Universal Robots PolyScope program: punto3_pickplace_NEW.urp

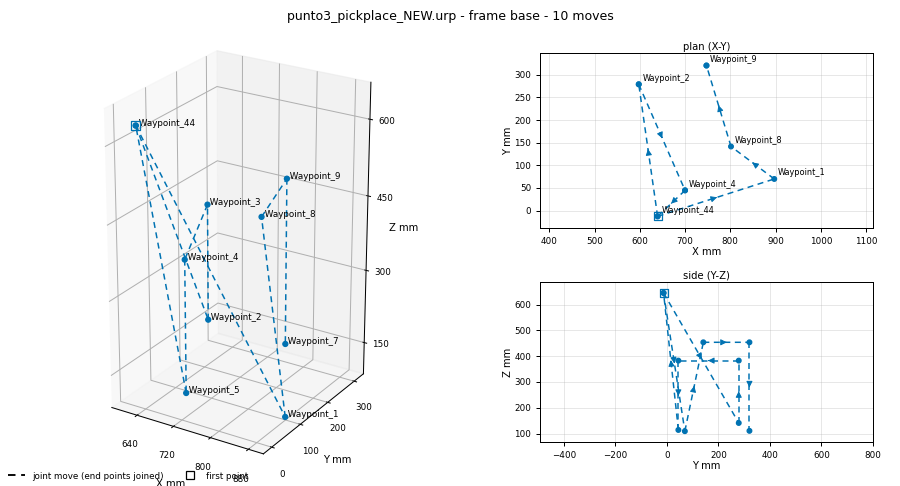
[picture p0: tool path of punto3_pickplace_NEW.urp in frame base, 10 of 10 moves have a stored position in this frame; points joined in program order, loops and branches not executed]
Program punto3_pickplace (installation=default directory=/ursim/programs createdIn=3.15.8.106339 lastSavedIn=3.15.8.106339 robotSerialNumber=2018359999)
Calibrated DH parameters: a=[0, -0.425, -0.39225, 0, 0, 0]; d=[0.089159, 0, 0, 0.10915, 0.09465, 0.0823]; alpha=[1.570796, 0, 0, 1.570796, -1.570796, 0]; deltaTheta=[0, 0, 0, 0, 0, 0]
Robot Program (runOnlyOnce=false)
  MoveJ speed 60 deg/s, acceleration 80 deg/s^2 (useActiveTCP=true)
    Set DigitalOutput pin=digital_out[0]; digitalValue=0
    Waypoint Waypoint_44: TCP in base x=639.374 y=-12.799 z=645.611 mm, rx=2.7019 ry=1.4477 rz=0.2985 rad; joints [8.631, -138.345, 17.122, 222.891, 90.378, -137.696] deg
    Wait DigitalInput pin=digital_in[0]; digitalValue=1
    Wait Sleep waitTime=2
    Waypoint Waypoint_2: TCP in base x=597.72 y=279.007 z=140.951 mm, rx=2.7019 ry=1.4477 rz=0.2985 rad; joints [35.16, -123.066, -94.887, 318.588, 85.157, -111.657] deg
    Set DigitalOutput pin=digital_out[0]; digitalValue=1
    Popup Message (haltProgram=false message=se cerró el gripper  inputType=Text)
    Waypoint Waypoint_3: TCP in base x=597.72 y=279.007 z=383.015 mm, rx=2.7019 ry=1.4477 rz=0.2985 rad; joints [35.16, -110.812, -75.083, 286.529, 85.157, -111.657] deg
    Popup Message (haltProgram=false message=punto intermedio principal inputType=Text)
    Wait Sleep waitTime=1
    Waypoint Waypoint_4: TCP in base x=700.042 y=44.656 z=383.015 mm, rx=2.7019 ry=1.4477 rz=0.2985 rad; joints [12.653, -116.851, -66.636, 285.153, 89.564, -133.757] deg
    Popup Message (haltProgram=false message=punto intermedio secundario inputType=Text)
    Wait Sleep waitTime=1
    Waypoint Waypoint_5: TCP in base x=700.042 y=44.656 z=113.852 mm, rx=2.7019 ry=1.4477 rz=0.2985 rad; joints [12.653, -129.957, -87.698, 319.32, 89.564, -133.757] deg
    Set DigitalOutput pin=digital_out[0]; digitalValue=0
    Popup Message (haltProgram=false message=se abrió el gripper inputType=Text)
    Waypoint Waypoint_44: TCP in base x=639.374 y=-12.799 z=645.611 mm, rx=2.7019 ry=1.4477 rz=0.2985 rad; joints [8.631, -138.345, 17.122, 222.891, 90.378, -137.696] deg
    Wait Sleep waitTime=2
    Waypoint Waypoint_1: TCP in base x=897.17 y=69.826 z=109 mm, rx=2.7019 ry=1.4477 rz=0.2985 rad; joints [11.435, -159.34, -30.741, 291.753, 89.811, -134.95] deg
    Set DigitalOutput pin=digital_out[0]; digitalValue=1
    Popup Message (haltProgram=false message=se cerró el gripper inputType=Text)
    Waypoint Waypoint_8: TCP in base x=801.574 y=141.533 z=454.057 mm, rx=2.7019 ry=1.4477 rz=0.2985 rad; joints [17.872, -148.017, -1.091, 250.688, 88.512, -128.645] deg
    Popup Message (haltProgram=false message=punto intermedio inicial inputType=Text)
    Waypoint Waypoint_9: TCP in base x=747.352 y=320.49 z=454.05 mm, rx=2.7019 ry=1.4477 rz=0.2985 rad; joints [31.347, -148.382, -0.155, 249.465, 85.871, -115.414] deg
    Popup Message (haltProgram=false message=punto intermedio secundario  inputType=Text)
    Wait Sleep waitTime=1
    Waypoint Waypoint_7: TCP in base x=747.352 y=320.49 z=110.361 mm, rx=2.7019 ry=1.4477 rz=0.2985 rad; joints [31.347, -143.617, -61.782, 306.327, 85.871, -115.414] deg
    Set DigitalOutput pin=digital_out[0]; digitalValue=0
    Popup Message (haltProgram=false message=se abrió el gripper inputType=Text)
    Wait Sleep waitTime=1
    Wait DigitalInput pin=digital_in[0]; digitalValue=1
